PROGRAM MAIN_2
VAR
	test2	: DINT;
END_VAR

test2:=test2+1;

END_PROGRAM

(* stored: Version 1.1.0.1, ProductVersion 3.1.4024.12
   POU MAIN_2: Id {0f2bedc6-1dcf-469e-aaf2-78b3082ce594}, SpecialFunc None *)
